{attribute 'GeneratedUsingTerminal: EL5112-0000-0016'}
{attribute addProperty BoxType "EL5112-0000-0016"}
{attribute addProperty Id "EtcSlaveTerminalBaseENC_Status_Channel_1AT %I*ENC_Status_Channel_10A67E5232ENC_Control_Channel_1AT %Q*ENC_Control_Channel_4C8A739514WcStateAT %I*WcState_9091E0EB2InfoDataAT %I*InfoData_32EB74EA10"}
{attribute addProperty CRC "2218874529"}
{attribute addProperty Size "58"}
TYPE EL5112_844156A1 EXTENDS EtcSlaveTerminalBase :
STRUCT
	{attribute addProperty Name "ENC_Status_Channel_1"}
	ENC_Status_Channel_1 : ENC_Status_Channel_10A67E52;
	{attribute addProperty Name "ENC_Control_Channel_1"}
	ENC_Control_Channel_1 : ENC_Control_Channel_4C8A7395;
	{attribute addProperty Name "WcState"}
	WcState : WcState_9091E0EB;
	{attribute addProperty Name "InfoData"}
	InfoData : InfoData_32EB74EA;
END_STRUCT
END_TYPE

(* stored: Version 1.2.0.0, ProductVersion 3.1.4024.9
   DUT EL5112_844156A1: Id {83b30e3c-c501-48dd-bcc3-823a88fb47ec} *)
